// TIA Portal V16 export
// export: Created 2021-09-08T12:46:09.1443302Z, ExportSetting WithDefaults, DisplayName Totally Integrated Automation Portal, DisplayVersion V16 Update 3, DisplayName TIA Portal Version Control Interface, DisplayVersion V16 Update 2, DisplayName TIA Portal Openness, DisplayVersion V16 Update 3, DisplayName TIA Portal Teamcenter Gateway, DisplayVersion V16, DisplayName STEP 7 Professional, DisplayVersion V16 Update 3, DisplayName STEP 7 Safety, DisplayVersion V16, DisplayName WinCC Advanced, DisplayVersion V16 Update 3
FUNCTION "AnalogHandler" : Void   // FC1, FBD
{ S7_Optimized_Access := 'TRUE' }
VERSION : 0.1
// stored: AutoNumber true, IsIECCheckEnabled false, SetENOAutomatically false, UDAEnableTagReadback false
   VAR_INPUT
      Ack : Bool;
      Piw : Array[*] of Int;
   END_VAR
   VAR_IN_OUT
      Data : Array[*] of "Ai";
   END_VAR
   VAR_TEMP
      tLb : Int;
      tUb : Int;
      i : Int;
   END_VAR
   VAR CONSTANT
      ERROR : Word := 16#01;
      BAD_PARAMETRS : Word := 16#02;
      HARDWARE_FAULT : Word := 16#04;
      SIMULATION : Word := 16#08;
      EMERGENCY_MIN : Word := 16#10;
      WARNING_MIN : Word := 16#20;
      WARNING_MAX : Word := 16#40;
      EMERGENCY_MAX : Word := 16#80;
   END_VAR
BEGIN

REGION Network 1 (SCL)
   #tLb := DINT_TO_INT(LOWER_BOUND(ARR := #Data, DIM := 1));
   #tUb := DINT_TO_INT(UPPER_BOUND(ARR := #Data, DIM := 1));

   FOR #i := #tLb TO #tUb DO
       #Data[#i].Par_code := #Piw[#i];
       #Data[#i].Par_mA := 4.0 + 16.0 * INT_TO_REAL(#Data[#i].Par_code) / 27648.0;

       IF #Data[#i].SimEnable THEN
           #Data[#i].badParam := #Data[#i].wireBreak := #Data[#i].overFlow := FALSE;
       ELSE
           #Data[#i].badParam := #Data[#i].rngUpLm < #Data[#i].rngLwLm;
           #Data[#i].wireBreak := #Data[#i].Par_code < -4866;//1.185 mA
           #Data[#i].overFlow := #Data[#i].Par_code > 32511; //22.81 mA
       END_IF;
       #Data[#i].Err :=
       #Data[#i].badParam OR
       #Data[#i].wireBreak OR
       #Data[#i].overFlow;

       IF #Data[#i].SimEnable THEN
           #Data[#i].Par := #Data[#i].SimValue;
       ELSE
           IF NOT #Data[#i].Err THEN
               #Data[#i].Par := #Data[#i].rngLwLm + INT_TO_REAL(#Data[#i].Par_code) * (#Data[#i].rngUpLm - #Data[#i].rngLwLm) / 27648.0;
               IF #Data[#i].disableParLessZero AND #Data[#i].Par < 0.0 THEN
                   #Data[#i].Par := 0.0;
               END_IF;
           ELSE
               #Data[#i].Par := 0;
           END_IF;
       END_IF;
       //Flags
       IF #Data[#i].Err THEN
           "setFlags"(enCondition := FALSE,
                      condition := #Data[#i].Par < #Data[#i].emrMin,
                      setTimerVal := #Data[#i].emrMinTime,
                      curFlag := #Data[#i].curEmMin,
                      mainFlag := #Data[#i].emMin,
                      timerVal := #Data[#i].curTimeEmrMin);
           "setFlags"(enCondition := FALSE,
                      condition := #Data[#i].Par > #Data[#i].emrMax,
                      setTimerVal := #Data[#i].emrMaxTime,
                      curFlag := #Data[#i].curEmMax,
                      mainFlag := #Data[#i].emMax,
                      timerVal := #Data[#i].curTimeEmrMax);
           "setFlags"(enCondition := FALSE,
                      condition := #Data[#i].Par < #Data[#i].wrnMin,
                      setTimerVal := #Data[#i].wrnMinTime,
                      curFlag := #Data[#i].curWnMin,
                      mainFlag := #Data[#i].wnMin,
                      timerVal := #Data[#i].curTimeWrnMin);
           "setFlags"(enCondition := FALSE,
                      condition := #Data[#i].Par > #Data[#i].wrnMax,
                      setTimerVal := #Data[#i].wrnMaxTime,
                      curFlag := #Data[#i].curWnMax,
                      mainFlag := #Data[#i].wnMax,
                      timerVal := #Data[#i].curTimeWrnMax);
           ELSE
           "setFlags"(enCondition:=#Data[#i].emMin_En,
                      condition:=#Data[#i].Par < #Data[#i].emrMin,
                      setTimerVal:=#Data[#i].emrMinTime,
                      curFlag:=#Data[#i].curEmMin,
                      mainFlag:=#Data[#i].emMin,
                      timerVal:=#Data[#i].curTimeEmrMin);
           "setFlags"(enCondition := #Data[#i].emMax_En,
                      condition := #Data[#i].Par > #Data[#i].emrMax,
                      setTimerVal := #Data[#i].emrMaxTime,
                      curFlag := #Data[#i].curEmMax,
                      mainFlag := #Data[#i].emMax,
                      timerVal := #Data[#i].curTimeEmrMax);
           "setFlags"(enCondition := #Data[#i].wrnMin_En,
                      condition := #Data[#i].Par < #Data[#i].wrnMin,
                      setTimerVal := #Data[#i].wrnMinTime,
                      curFlag := #Data[#i].curWnMin,
                      mainFlag := #Data[#i].wnMin,
                      timerVal := #Data[#i].curTimeWrnMin);
           "setFlags"(enCondition := #Data[#i].wrnMax_En,
                      condition := #Data[#i].Par > #Data[#i].wrnMax,
                      setTimerVal := #Data[#i].wrnMaxTime,
                      curFlag := #Data[#i].curWnMax,
                      mainFlag := #Data[#i].wnMax,
                      timerVal := #Data[#i].curTimeWrnMax);
       END_IF;
       //Ack
   //    #Data[#i].ackAll := #Ack;
       IF #Data[#i].modeAck THEN
           IF #Data[#i].ackAll THEN
               #Data[#i].emMin := #Data[#i].emMax := #Data[#i].wnMin := #Data[#i].wnMax := FALSE;
               #Data[#i].curTimeEmrMin := #Data[#i].curTimeEmrMax := #Data[#i].curTimeWrnMin := #Data[#i].curTimeWrnMax := 0;
           END_IF;
           IF (#Data[#i].ack AND 16#10) > 0 THEN
               #Data[#i].emMin := FALSE;
               #Data[#i].curTimeEmrMin := 0;
               #Data[#i].ack := #Data[#i].ack AND NOT(DWORD_TO_BYTE(#EMERGENCY_MIN));
           END_IF;
           IF (#Data[#i].ack AND 16#80) > 0 THEN
               #Data[#i].emMax := FALSE;
               #Data[#i].curTimeEmrMax := 0;
               #Data[#i].ack := #Data[#i].ack AND NOT(DWORD_TO_BYTE(#EMERGENCY_MAX));
           END_IF;
       ELSE
           IF NOT #Data[#i].curEmMin THEN
               #Data[#i].emMin := FALSE;
           END_IF;
           IF NOT #Data[#i].curEmMax THEN
               #Data[#i].emMax := FALSE;
           END_IF;
       END_IF;
       //Rst warning flags after normalization value
       IF NOT #Data[#i].curWnMin THEN
           #Data[#i].wnMin := FALSE;
       END_IF;
       IF NOT #Data[#i].curWnMax THEN
           #Data[#i].wnMax := FALSE;
       END_IF;
       //States:
       "setState"(condition:= NOT #Data[#i].Err,
                  hexVal:=#ERROR,
                  state:=#Data[#i].State);
       "setState"(condition := #Data[#i].badParam,
                  hexVal := #BAD_PARAMETRS,
                  state := #Data[#i].State);
       "setState"(condition := #Data[#i].wireBreak OR #Data[#i].overFlow,
                  hexVal := #HARDWARE_FAULT,
                  state := #Data[#i].State);
       "setState"(condition := #Data[#i].SimEnable,
                  hexVal := #SIMULATION,
                  state := #Data[#i].State);
       "setState"(condition := #Data[#i].emMin,
                  hexVal := #EMERGENCY_MIN,
                  state := #Data[#i].State);
       "setState"(condition := #Data[#i].wnMin,
                  hexVal := #WARNING_MIN,
                  state := #Data[#i].State);
       "setState"(condition := #Data[#i].wnMax,
                  hexVal := #WARNING_MAX,
                  state := #Data[#i].State);
       "setState"(condition := #Data[#i].emMax,
                  hexVal := #EMERGENCY_MAX,
                  state := #Data[#i].State);
   END_FOR;
END_REGION
END_FUNCTION
